TYPE ST_4PViciValveSampleNames :
STRUCT
      {attribute 'pytmc' := '
        pv: 01
        io: io
        autosave_pass0: VAL DESC
     '}
     s1 : STRING;
     {attribute 'pytmc' := '
        pv: 02
        io: io
        autosave_pass0: VAL DESC
     '}
     s2 : STRING;
     {attribute 'pytmc' := '
        pv: 03
        io: io
        autosave_pass0: VAL DESC
     '}
     s3 : STRING;
     {attribute 'pytmc' := '
        pv: 04
        io: io
        autosave_pass0: VAL DESC
     '}
     s4 : STRING;
END_STRUCT
END_TYPE

(* stored: Version 1.1.0.1, ProductVersion 3.1.4024.12
   DUT ST_4PViciValveSampleNames: Id {35be0b4c-67ce-4822-bad8-6de307e4269c} *)
